// TIA Portal V17 export
// export: Created 2024-06-14T09:52:29.4394536Z, ExportSetting WithDefaults, DisplayName Totally Integrated Automation Portal, DisplayVersion V17, DisplayName TIA Portal Openness, DisplayVersion V17, DisplayName TIA Portal Version Control Interface, DisplayVersion V17, DisplayName Simotion SCOUT TIA, DisplayVersion 5.4.3.0, DisplayName SINAMICS Startdrive Advanced, DisplayVersion V17 SP1 Update 1, DisplayName SINAMICS Startdrive G110M, G120, G120C, G120D, G120P, G115D, DisplayVersion V17 SP1 Update 1, DisplayName SINAMICS Startdrive G130, G150, S120, S150, SINAMICS MV, S210, DisplayVersion V17 SP1 Update 1, DisplayName STEP 7 Professional, DisplayVersion V17, DisplayName STEP 7 Safety, DisplayVersion V17, DisplayName WinCC Professional, DisplayVersion V17
DATA_BLOCK "TCP_STN4_STN1_FB_DB"   // DB110
VERSION : 0.1
// stored: AutoNumber false, DBAccessibleFromOPCUA true, InstanceOfName TCP_STN4_STN1_FB, InstanceOfType FB
"TCP_STN4_STN1_FB"
   // VAR_OUTPUT
   //    Modbus_Busy : Bool;
   // END_VAR
   // VAR_IN_OUT
   //    Mod_TCP_Setup : "Mod_TCP_Data";
   //    LPG_Fill_Data : "LPG_FILL_DATA";
   // END_VAR
   // VAR
   //    PStep_No : Struct
   //       MASTER_STEP_NO : "Master_Step_No";
   //    END_STRUCT;
   //    Write_Bit_Address : Int;
   //    TRIG : Array[1..100] of Bool;
   //    MOD_MASTER1_REQ : Array[1..10] of Bool;
   //    MOD_MASTER2_REQ : Array[1..10] of Bool;
   //    MOD_MASTER3_REQ : Array[1..10] of Bool;
   //    MOD_MASTER4_REQ : Array[1..10] of Bool;
   //    MOD_MASTER5_REQ : Array[1..10] of Bool;
   //    MOD_MASTER6_REQ : Array[1..10] of Bool;
   //    MAS_TRG_EXTN { S7_SetPoint := 'True'} : TOF_TIME;
   //    Tare_delay { S7_SetPoint := 'True'} : TON_TIME;
   // END_VAR
BEGIN
END_DATA_BLOCK
